FUNCTION_BLOCK FB_ConvertColourSpace
VAR_INPUT
	hr_internal			: HRESULT; 
	ipImageIn		: ITcVnImage; //Only takes RGB
	ColourSpaceType	:STRING; // Only HSV or GRAY for now
END_VAR
VAR_OUTPUT
	ipImageOut		: ITcVnImage;
END_VAR
VAR
	GRAY	:STRING := 'GRAY';
	HSV		:STRING := 'HSV';
END_VAR

IF ColourSpaceType = 'GRAY' THEN
	hr_internal	:= F_VN_ConvertColorSpace(ipImageIn, ipImageOut, TCVN_CST_RGB_TO_GRAY, hr_internal	);
ELSIF ColourSpaceType = 'HSV' THEN
	hr_internal	 := F_VN_ConvertColorSpace(ipImageIn, ipImageOut, TCVN_CST_RGB_TO_HSV, hr_internal	);
END_IF

END_FUNCTION_BLOCK

(* stored: Version 1.1.0.1, ProductVersion 3.1.4024.12
   POU FB_ConvertColourSpace: Id {d94bcad0-66b2-4a3a-8115-2088d66c5adb}, SpecialFunc None *)
